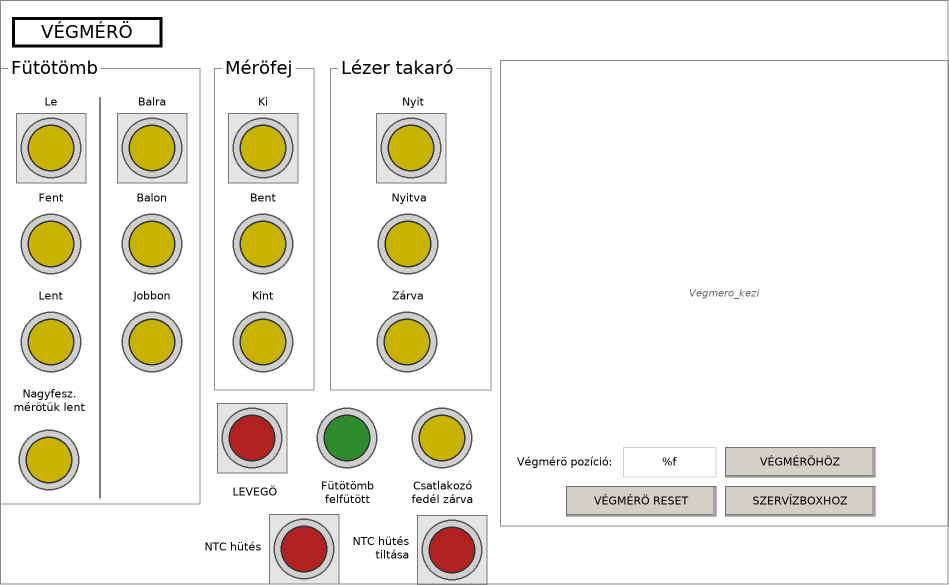
VISUALIZATION Vegmero  // 949x585
    Lamp1 (407,403 70x70), variable: VEGMERO.bFedelNyitva, style: Lamp-Lamp1-Yellow
    Label (405,478 75x29), "Csatlakozó fedél zárva"
    GroupBox (0,60 200x444), "Fütötömb"
        Lamp1 (16,247 70x70), variable: VEGMERO.bPlatniLent, style: Lamp-Lamp1-Yellow
        Label (26,226 50x20), "Lent"
        PushSwitch (16,53 70x70), variable: VEGMERO.bPlatniFelLe, behaviour: TOGGLE, style: Switch-PushSwitch-Yellow
        Label (26,32 50x20), "Le"
        Lamp1 (16,149 70x70), variable: VEGMERO.bPlatniFent, style: Lamp-Lamp1-Yellow
        Label (26,128 50x20), "Fent"
        Lamp1 (117,149 70x70), variable: VEGMERO.bPlatniBalon, style: Lamp-Lamp1-Yellow
        Label (127,128 50x20), "Balon"
        Lamp1 (117,247 70x70), variable: VEGMERO.bPlatniJobbon, style: Lamp-Lamp1-Yellow
        Label (127,226 50x20), "Jobbon"
        PushSwitch (117,53 70x70), variable: VEGMERO.bPlatniBalraJobbra, behaviour: TOGGLE, style: Switch-PushSwitch-Yellow
        Label (127,32 50x20), "Balra"
        Line (100,438) (100,37)
        Label (8,323 83x35), "Nagyfesz. mérötük lent"
        Lamp1 (14,365 70x70), variable: VEGMERO.bNagyFeszMerotuLent, style: Lamp-Lamp1-Yellow
    GroupBox (214,60 100x330), "Méröfej"
        Lamp1 (14,149 70x70), variable: VEGMERO.bMerotukBent, style: Lamp-Lamp1-Yellow
        Label (24,128 50x20), "Bent"
        Lamp1 (14,247 70x70), variable: VEGMERO.bMerotukKint, style: Lamp-Lamp1-Yellow
        Label (24,226 50x20), "Kint"
        PushSwitch (14,53 70x70), variable: VEGMERO.bMerotukBeKi, behaviour: TOGGLE, style: Switch-PushSwitch-Yellow
        Label (24,32 50x20), "Ki"
    GroupBox (330,60 161x330), "Lézer takaró"
        PushSwitch (46,53 70x70), variable: VEGMERO.bLezertakaro, behaviour: TOGGLE, style: Switch-PushSwitch-Yellow
        Label (58,32 50x20), "Nyit"
        Lamp1 (43,149 70x70), variable: VEGMERO.bLezertakaroNyitva, style: Lamp-Lamp1-Yellow
        Label (54,128 50x20), "Nyitva"
        Lamp1 (42,247 70x70), variable: VEGMERO.bLezertakaroZarva, style: Lamp-Lamp1-Yellow
        Label (53,226 50x20), "Zárva"
    TabControl (500,60 449x466)
        shows Vegmero_kezi()
        shows Vegmero_auto()
        [0]: TabTitle=Kézi
        [1]: TabTitle=Automata
    RoundedRectangle (12,17 150x30)
    Label (12,17 150x30), "VÉGMÉRÖ"
    Label (511,452 104x20), "Végmérö pozíció:"
    Textfield (623,447 93x30), "%f", text variable: GVL.lrVegmeroPosition
        OnMouseClick: write the text variable via VisuDialogs.Numpad, min -10000, max -1
    Button (725,447 150x30), "VÉGMÉRÖHÖZ"
        OnMouseUp: execute { PISTITENGELY.lrPistiPosition:=GVL.lrVegmeroPosition; PISTITENGELY.sPistiAxisCommand:='MOVE'; }
    Lamp1 (312,403 70x70), variable: GVL.bHeatingTempOK, style: Lamp-Lamp1-Green
    Label (310,478 75x29), "Fütötömb felfütött"
    Group (217,403 70x104)
        PushSwitch (0,0 70x70), variable: MAIN.bLevego, behaviour: TOGGLE, style: Switch-PushSwitch-Red
        Label (8,74 55x30), "LEVEGÖ"
    Button (725,486 150x30), "SZERVÍZBOXHOZ"
        OnMouseUp: execute { PISTITENGELY.lrPistiPosition:=GVL.lrPtSzervizbox; PISTITENGELY.sPistiAxisCommand:='MOVE'; }
    Button (566,486 150x30), "VÉGMÉRÖ RESET"
        OnMouseUp: execute { VEGMERO.iState:=0; VEGMERO.s_InCommand:='RESET'; }
    PushSwitch (269,514 70x70), variable: VEGMERO.bKeziHutes, behaviour: TOGGLE, style: Switch-PushSwitch-Red
    Label (196,532 68x30), "NTC hütés"
    PushSwitch (417,515 70x70), variable: VEGMERO.bHutesTiltas, behaviour: TOGGLE, style: Switch-PushSwitch-Red
    Label (344,533 68x30), "NTC hütés tiltása"
END_VISUALIZATION

(* stored: Version 1.1.0.1, ProductVersion 3.1.4024.11
   Visu Vegmero: Id {fd71e4b0-da89-4d0b-a63e-e3ed1029a8e6} *)
